(* ---------------------------------------------------------
   Z轴External纯轨迹发生器。
   进入：External Adapter已Active且已接受P/V/A/Direction有效。
   周期动作：只从最后accepted包进行Rate Limit和梯形积分。
   换向：零速、旧方向保持、方向归零、新方向预置均由accepted Feed推进。
   硬禁止：同一扫描保持accepted位置并发布V=0、A=0、方向不变。
   Fault：首次故障锁存；调用者必须停止Feed并请求Adapter安全Disable。
   --------------------------------------------------------- *)
stOutput.rPosition_mm := 0.0;
stOutput.rVelocity_mm_s := 0.0;
stOutput.rAcceleration_mm_s2 := 0.0;
stOutput.nDirection := 0;
stOutput.eState := eState;
stOutput.bDirectionTransition := FALSE;
stOutput.bZeroConfirmed := FALSE;
stOutput.bPositiveMotionInhibited := FALSE;
stOutput.bActive := FALSE;
stOutput.bFault := bFaultLatched;
stOutput.nFaultId := udiLatchedFaultId;

(* Fault只能在未使能时显式复位；复位扫描保持IDLE和非活动。 *)
IF bFaultLatched THEN
    eState := Z_TRAJ_FAULT;
    stOutput.eState := Z_TRAJ_FAULT;
    stOutput.bActive := FALSE;
    stOutput.bFault := TRUE;
    stOutput.nFaultId := udiLatchedFaultId;
    IF stInput.bReset AND NOT stInput.bEnable THEN
        bFaultLatched := FALSE;
        udiLatchedFaultId := 0;
        bInitialized := FALSE;
        bLastPublishedPositiveMotionInhibited := FALSE;
        udiLastAcceptedFeedCycleCounter := 0;
        nLastNonZeroDirection := 0;
        nPendingDirection := 0;
        nAcceptedStateCycles := 0;
        eState := Z_TRAJ_IDLE;
        stOutput.bFault := FALSE;
        stOutput.nFaultId := 0;
        stOutput.bActive := FALSE;
        stOutput.eState := Z_TRAJ_IDLE;
    END_IF;
    RETURN;
END_IF;

(* Disable清除运行态但不伪造Active或轨迹Feed。 *)
IF NOT stInput.bEnable THEN
    bInitialized := FALSE;
    bLastPublishedPositiveMotionInhibited := FALSE;
    udiLastAcceptedFeedCycleCounter := 0;
    nLastNonZeroDirection := 0;
    nPendingDirection := 0;
    nAcceptedStateCycles := 0;
    eState := Z_TRAJ_IDLE;
    stOutput.eState := Z_TRAJ_IDLE;
    RETURN;
END_IF;

nTargetDirection := 0;
IF stInput.rTargetVelocity_mm_s > 0.0 THEN
    nTargetDirection := 1;
ELSIF stInput.rTargetVelocity_mm_s < 0.0 THEN
    nTargetDirection := -1;
END_IF;

bConfigurationValid := (stInput.rCycleTime_s > 0.0)
    AND FC_IsFiniteLReal(rValue := stInput.rCycleTime_s)
    AND FC_IsFiniteLReal(rValue := stInput.rMinimumPosition_mm)
    AND FC_IsFiniteLReal(rValue := stInput.rMaximumPosition_mm)
    AND (stInput.rMaximumPosition_mm > stInput.rMinimumPosition_mm)
    AND FC_IsFiniteLReal(rValue := stInput.rMaximumVelocity_mm_s)
    AND (stInput.rMaximumVelocity_mm_s > 0.0)
    AND FC_IsFiniteLReal(rValue := stInput.rMaximumAcceleration_mm_s2)
    AND (stInput.rMaximumAcceleration_mm_s2 > 0.0)
    AND FC_IsFiniteLReal(rValue := stInput.rStandstillVelocity_mm_s)
    AND (stInput.rStandstillVelocity_mm_s >= 0.0)
    AND (stInput.rStandstillVelocity_mm_s < stInput.rMaximumVelocity_mm_s)
    AND FC_IsFiniteLReal(rValue := stInput.rMaximumPositionDeviation_mm)
    AND (stInput.rMaximumPositionDeviation_mm >= 0.0)
    AND FC_IsFiniteLReal(rValue := stInput.rTargetVelocity_mm_s)
    AND (ABS(stInput.rTargetVelocity_mm_s) <= stInput.rMaximumVelocity_mm_s)
    AND (stInput.nDirectionHoldCycles >= 1);

IF NOT bConfigurationValid THEN
    bFaultLatched := TRUE;
    udiLatchedFaultId := 16#0000B001;
    eState := Z_TRAJ_FAULT;
    stOutput.bFault := TRUE;
    stOutput.nFaultId := udiLatchedFaultId;
    stOutput.eState := Z_TRAJ_FAULT;
    stOutput.bActive := FALSE;
    RETURN;
END_IF;

(* Adapter未Active时只等待重新同步，不消费或外推任何包。 *)
IF stInput.eExternalState <> Z_EXT_ACTIVE THEN
    bInitialized := FALSE;
    bLastPublishedPositiveMotionInhibited := FALSE;
    nAcceptedStateCycles := 0;
    eState := Z_TRAJ_SYNC;
    stOutput.eState := Z_TRAJ_SYNC;
    RETURN;
END_IF;

bAcceptedMotionValid := stInput.bAcceptedSetpointValid
    AND FC_IsFiniteLReal(rValue := stInput.rAcceptedPosition_mm)
    AND FC_IsFiniteLReal(rValue := stInput.rAcceptedVelocity_mm_s)
    AND FC_IsFiniteLReal(rValue := stInput.rAcceptedAcceleration_mm_s2)
    AND (ABS(stInput.rAcceptedVelocity_mm_s) <= stInput.rMaximumVelocity_mm_s)
    AND (ABS(stInput.rAcceptedAcceleration_mm_s2) <= stInput.rMaximumAcceleration_mm_s2);

IF NOT bAcceptedMotionValid THEN
    bFaultLatched := TRUE;
    udiLatchedFaultId := 16#0000B002;
    eState := Z_TRAJ_FAULT;
    stOutput.bFault := TRUE;
    stOutput.nFaultId := udiLatchedFaultId;
    stOutput.eState := Z_TRAJ_FAULT;
    stOutput.bActive := FALSE;
    RETURN;
END_IF;

IF (stInput.nAcceptedDirection < -1) OR (stInput.nAcceptedDirection > 1) THEN
    bFaultLatched := TRUE;
    udiLatchedFaultId := 16#0000B003;
    eState := Z_TRAJ_FAULT;
    stOutput.bFault := TRUE;
    stOutput.nFaultId := udiLatchedFaultId;
    stOutput.eState := Z_TRAJ_FAULT;
    stOutput.bActive := FALSE;
    RETURN;
END_IF;

IF (stInput.rAcceptedPosition_mm < stInput.rMinimumPosition_mm)
    OR (stInput.rAcceptedPosition_mm > stInput.rMaximumPosition_mm) THEN
    bFaultLatched := TRUE;
    udiLatchedFaultId := 16#0000B004;
    eState := Z_TRAJ_FAULT;
    stOutput.bFault := TRUE;
    stOutput.nFaultId := udiLatchedFaultId;
    stOutput.eState := Z_TRAJ_FAULT;
    stOutput.bActive := FALSE;
    RETURN;
END_IF;

IF (stInput.nAcceptedDirection = 0)
    AND ((ABS(stInput.rAcceptedVelocity_mm_s) > stInput.rStandstillVelocity_mm_s)
        OR (stInput.rAcceptedAcceleration_mm_s2 <> 0.0)) THEN
    bFaultLatched := TRUE;
    udiLatchedFaultId := 16#0000B007;
    eState := Z_TRAJ_FAULT;
    stOutput.bFault := TRUE;
    stOutput.nFaultId := udiLatchedFaultId;
    stOutput.eState := Z_TRAJ_FAULT;
    stOutput.bActive := FALSE;
    RETURN;
END_IF;

IF ((stInput.rAcceptedVelocity_mm_s > stInput.rStandstillVelocity_mm_s)
        AND (stInput.nAcceptedDirection <> 1))
    OR ((stInput.rAcceptedVelocity_mm_s < -stInput.rStandstillVelocity_mm_s)
        AND (stInput.nAcceptedDirection <> -1)) THEN
    bFaultLatched := TRUE;
    udiLatchedFaultId := 16#0000B006;
    eState := Z_TRAJ_FAULT;
    stOutput.bFault := TRUE;
    stOutput.nFaultId := udiLatchedFaultId;
    stOutput.eState := Z_TRAJ_FAULT;
    stOutput.bActive := FALSE;
    RETURN;
END_IF;

bNewAcceptedFeed := (stInput.bFeedAccepted = TRUE)
    AND (stInput.udiAcceptedFeedCycleCounter <> udiLastAcceptedFeedCycleCounter);
bAcceptedPublishedZero := FALSE;
stOutput.bPositiveMotionInhibited := stInput.bInhibitPositiveMotion;

IF NOT bInitialized THEN
    (* 首个Active扫描只发布同步包；必须等该包accepted后才进入TRACKING。 *)
    udiLastAcceptedFeedCycleCounter := stInput.udiAcceptedFeedCycleCounter;
    IF stInput.nAcceptedDirection <> 0 THEN
        nLastNonZeroDirection := stInput.nAcceptedDirection;
    END_IF;
    bInitialized := TRUE;
    eState := Z_TRAJ_SYNC;
    stOutput.eState := Z_TRAJ_SYNC;
    stOutput.rPosition_mm := stInput.rAcceptedPosition_mm;
    stOutput.rVelocity_mm_s := stInput.rAcceptedVelocity_mm_s;
    stOutput.rAcceleration_mm_s2 := stInput.rAcceptedAcceleration_mm_s2;
    stOutput.nDirection := stInput.nAcceptedDirection;
    IF stInput.bInhibitPositiveMotion
        AND (stInput.rAcceptedVelocity_mm_s > 0.0) THEN
        stOutput.rPosition_mm := stInput.rAcceptedPosition_mm;
        stOutput.rVelocity_mm_s := 0.0;
        stOutput.rAcceleration_mm_s2 := 0.0;
        stOutput.nDirection := stInput.nAcceptedDirection;
        stOutput.bPositiveMotionInhibited := TRUE;
    END_IF;
    rLastPublishedPosition_mm := stOutput.rPosition_mm;
    rLastPublishedVelocity_mm_s := stOutput.rVelocity_mm_s;
    rLastPublishedAcceleration_mm_s2 := stOutput.rAcceleration_mm_s2;
    nLastPublishedDirection := stOutput.nDirection;
    bLastPublishedPositiveMotionInhibited := stOutput.bPositiveMotionInhibited;
    stOutput.bActive := TRUE;
    RETURN;
ELSE
    IF bNewAcceptedFeed THEN
        IF (stInput.nAcceptedDirection <> nLastPublishedDirection)
            AND (ABS(stInput.rAcceptedVelocity_mm_s) > stInput.rStandstillVelocity_mm_s) THEN
            bFaultLatched := TRUE;
            udiLatchedFaultId := 16#0000B006;
            eState := Z_TRAJ_FAULT;
            stOutput.bFault := TRUE;
            stOutput.nFaultId := udiLatchedFaultId;
            stOutput.eState := Z_TRAJ_FAULT;
            stOutput.bActive := FALSE;
            RETURN;
        END_IF;
        IF (eState <> Z_TRAJ_PRELOAD_NEW_DIRECTION)
            AND (stInput.nAcceptedDirection <> 0)
            AND (nLastNonZeroDirection <> 0)
            AND (stInput.nAcceptedDirection <> nLastNonZeroDirection) THEN
            bFaultLatched := TRUE;
            udiLatchedFaultId := 16#0000B006;
            eState := Z_TRAJ_FAULT;
            stOutput.bFault := TRUE;
            stOutput.nFaultId := udiLatchedFaultId;
            stOutput.eState := Z_TRAJ_FAULT;
            stOutput.bActive := FALSE;
            RETURN;
        END_IF;

        bAcceptedContinuityValid := ABS(stInput.rAcceptedPosition_mm
                - rLastPublishedPosition_mm) <= stInput.rMaximumPositionDeviation_mm
            AND (stInput.rAcceptedVelocity_mm_s = rLastPublishedVelocity_mm_s)
            AND (stInput.rAcceptedAcceleration_mm_s2 = rLastPublishedAcceleration_mm_s2)
            AND (stInput.nAcceptedDirection = nLastPublishedDirection);
        IF NOT bAcceptedContinuityValid THEN
            bFaultLatched := TRUE;
            udiLatchedFaultId := 16#0000B005;
            eState := Z_TRAJ_FAULT;
            stOutput.bFault := TRUE;
            stOutput.nFaultId := udiLatchedFaultId;
            stOutput.eState := Z_TRAJ_FAULT;
            stOutput.bActive := FALSE;
            RETURN;
        END_IF;

        bAcceptedPublishedZero := (rLastPublishedVelocity_mm_s = 0.0)
            AND (rLastPublishedAcceleration_mm_s2 = 0.0)
            AND (ABS(stInput.rAcceptedVelocity_mm_s) <= stInput.rStandstillVelocity_mm_s)
            AND (stInput.rAcceptedAcceleration_mm_s2 = 0.0);
        udiLastAcceptedFeedCycleCounter := stInput.udiAcceptedFeedCycleCounter;
        IF stInput.nAcceptedDirection <> 0 THEN
            nLastNonZeroDirection := stInput.nAcceptedDirection;
        END_IF;
    END_IF;
END_IF;

stOutput.bZeroConfirmed := bNewAcceptedFeed AND bAcceptedPublishedZero;

(* 转换期间目标方向必须保持为进入转换时锁存的非零方向。 *)
IF (eState = Z_TRAJ_RAMP_TO_ZERO)
    OR (eState = Z_TRAJ_HOLD_OLD_DIRECTION)
    OR (eState = Z_TRAJ_DIRECTION_ZERO)
    OR (eState = Z_TRAJ_PRELOAD_NEW_DIRECTION) THEN
    IF (nTargetDirection = 0) OR (nTargetDirection <> nPendingDirection) THEN
        bFaultLatched := TRUE;
        udiLatchedFaultId := 16#0000B00A;
        eState := Z_TRAJ_FAULT;
        stOutput.bFault := TRUE;
        stOutput.nFaultId := udiLatchedFaultId;
        stOutput.eState := Z_TRAJ_FAULT;
        stOutput.bActive := FALSE;
        RETURN;
    END_IF;
END_IF;

stOutput.eState := eState;
stOutput.bDirectionTransition := (eState = Z_TRAJ_RAMP_TO_ZERO)
    OR (eState = Z_TRAJ_HOLD_OLD_DIRECTION)
    OR (eState = Z_TRAJ_DIRECTION_ZERO)
    OR (eState = Z_TRAJ_PRELOAD_NEW_DIRECTION);

(* Hard Inhibit是唯一允许替换未接受普通包的安全优先级。 *)
IF NOT bNewAcceptedFeed AND stInput.bInhibitPositiveMotion
    AND ((stInput.rAcceptedVelocity_mm_s > 0.0)
        OR (rLastPublishedVelocity_mm_s > 0.0)) THEN
    stOutput.rPosition_mm := stInput.rAcceptedPosition_mm;
    stOutput.rVelocity_mm_s := 0.0;
    stOutput.rAcceleration_mm_s2 := 0.0;
    stOutput.nDirection := stInput.nAcceptedDirection;
    stOutput.bPositiveMotionInhibited := TRUE;
    rLastPublishedPosition_mm := stOutput.rPosition_mm;
    rLastPublishedVelocity_mm_s := stOutput.rVelocity_mm_s;
    rLastPublishedAcceleration_mm_s2 := stOutput.rAcceleration_mm_s2;
    nLastPublishedDirection := stOutput.nDirection;
    bLastPublishedPositiveMotionInhibited := stOutput.bPositiveMotionInhibited;
    stOutput.bActive := TRUE;
    RETURN;
END_IF;

(* 无新accepted counter时严格重复待接受包，忽略TRACKING实时目标变化。 *)
IF NOT bNewAcceptedFeed THEN
    stOutput.rPosition_mm := rLastPublishedPosition_mm;
    stOutput.rVelocity_mm_s := rLastPublishedVelocity_mm_s;
    stOutput.rAcceleration_mm_s2 := rLastPublishedAcceleration_mm_s2;
    stOutput.nDirection := nLastPublishedDirection;
    stOutput.bPositiveMotionInhibited := bLastPublishedPositiveMotionInhibited;
    stOutput.bActive := TRUE;
    RETURN;
END_IF;

CASE eState OF
    Z_TRAJ_IDLE:
        eState := Z_TRAJ_SYNC;

    Z_TRAJ_SYNC:
        (* 同步扫描原样发布accepted包，下一扫描才开始积分。 *)
        stOutput.rPosition_mm := stInput.rAcceptedPosition_mm;
        stOutput.rVelocity_mm_s := stInput.rAcceptedVelocity_mm_s;
        stOutput.rAcceleration_mm_s2 := stInput.rAcceptedAcceleration_mm_s2;
        stOutput.nDirection := stInput.nAcceptedDirection;
        IF bInitialized THEN
            eState := Z_TRAJ_TRACKING;
        END_IF;

    Z_TRAJ_TRACKING:
        IF (nTargetDirection <> 0)
            AND (nLastNonZeroDirection <> 0)
            AND (nTargetDirection <> nLastNonZeroDirection) THEN
            (* 非零反向目标先按accepted速度主动降到零。 *)
            nPendingDirection := nTargetDirection;
            nAcceptedStateCycles := 0;
            eState := Z_TRAJ_RAMP_TO_ZERO;
            rNextVelocity_mm_s := FC_LimitRate(
                rCurrent := stInput.rAcceptedVelocity_mm_s,
                rTarget := 0.0,
                rRateUpPer_s := stInput.rMaximumAcceleration_mm_s2,
                rRateDownPer_s := stInput.rMaximumAcceleration_mm_s2,
                rCycleTime_s := stInput.rCycleTime_s);
            rNextAcceleration_mm_s2 :=
                (rNextVelocity_mm_s - stInput.rAcceptedVelocity_mm_s)
                / stInput.rCycleTime_s;
            rNextPosition_mm := stInput.rAcceptedPosition_mm
                + 0.5 * (stInput.rAcceptedVelocity_mm_s + rNextVelocity_mm_s)
                * stInput.rCycleTime_s;
            stOutput.rPosition_mm := rNextPosition_mm;
            stOutput.rVelocity_mm_s := rNextVelocity_mm_s;
            stOutput.rAcceleration_mm_s2 := rNextAcceleration_mm_s2;
            stOutput.nDirection := nLastNonZeroDirection;
        ELSIF (stInput.nAcceptedDirection = 0) AND (nTargetDirection <> 0) THEN
            (* 静止初始状态先预置新方向一个被接受的完整周期。 *)
            nPendingDirection := nTargetDirection;
            nAcceptedStateCycles := 0;
            eState := Z_TRAJ_PRELOAD_NEW_DIRECTION;
            stOutput.rPosition_mm := stInput.rAcceptedPosition_mm;
            stOutput.rVelocity_mm_s := 0.0;
            stOutput.rAcceleration_mm_s2 := 0.0;
            stOutput.nDirection := nPendingDirection;
        ELSE
            rNextVelocity_mm_s := FC_LimitRate(
                rCurrent := stInput.rAcceptedVelocity_mm_s,
                rTarget := stInput.rTargetVelocity_mm_s,
                rRateUpPer_s := stInput.rMaximumAcceleration_mm_s2,
                rRateDownPer_s := stInput.rMaximumAcceleration_mm_s2,
                rCycleTime_s := stInput.rCycleTime_s);
            IF stInput.bInhibitPositiveMotion AND (rNextVelocity_mm_s > 0.0) THEN
                rNextVelocity_mm_s := 0.0;
            END_IF;
            rNextAcceleration_mm_s2 :=
                (rNextVelocity_mm_s - stInput.rAcceptedVelocity_mm_s)
                / stInput.rCycleTime_s;
            rNextPosition_mm := stInput.rAcceptedPosition_mm
                + 0.5 * (stInput.rAcceptedVelocity_mm_s + rNextVelocity_mm_s)
                * stInput.rCycleTime_s;
            stOutput.rPosition_mm := rNextPosition_mm;
            stOutput.rVelocity_mm_s := rNextVelocity_mm_s;
            stOutput.rAcceleration_mm_s2 := rNextAcceleration_mm_s2;
            stOutput.nDirection := stInput.nAcceptedDirection;
        END_IF;

        (* Hard Force/Stroke/Collision覆盖普通正向制动尾巴。 *)
        IF stInput.bInhibitPositiveMotion THEN
            IF stInput.rAcceptedVelocity_mm_s > 0.0 THEN
                stOutput.rPosition_mm := stInput.rAcceptedPosition_mm;
                stOutput.rVelocity_mm_s := 0.0;
                stOutput.rAcceleration_mm_s2 := 0.0;
                stOutput.nDirection := stInput.nAcceptedDirection;
                stOutput.bPositiveMotionInhibited := TRUE;
            ELSIF stOutput.rVelocity_mm_s > 0.0 THEN
                stOutput.rPosition_mm := stInput.rAcceptedPosition_mm;
                stOutput.rVelocity_mm_s := 0.0;
                stOutput.rAcceleration_mm_s2 := 0.0;
                stOutput.nDirection := stInput.nAcceptedDirection;
                stOutput.bPositiveMotionInhibited := TRUE;
            ELSE
                stOutput.bPositiveMotionInhibited := TRUE;
            END_IF;
        END_IF;

    Z_TRAJ_RAMP_TO_ZERO:
        rNextVelocity_mm_s := FC_LimitRate(
            rCurrent := stInput.rAcceptedVelocity_mm_s,
            rTarget := 0.0,
            rRateUpPer_s := stInput.rMaximumAcceleration_mm_s2,
            rRateDownPer_s := stInput.rMaximumAcceleration_mm_s2,
            rCycleTime_s := stInput.rCycleTime_s);
        IF ABS(rNextVelocity_mm_s) <= stInput.rStandstillVelocity_mm_s THEN
            rNextVelocity_mm_s := 0.0;
        END_IF;
        rNextAcceleration_mm_s2 :=
            (rNextVelocity_mm_s - stInput.rAcceptedVelocity_mm_s)
            / stInput.rCycleTime_s;
        rNextPosition_mm := stInput.rAcceptedPosition_mm
            + 0.5 * (stInput.rAcceptedVelocity_mm_s + rNextVelocity_mm_s)
            * stInput.rCycleTime_s;
        stOutput.rPosition_mm := rNextPosition_mm;
        stOutput.rVelocity_mm_s := rNextVelocity_mm_s;
        stOutput.rAcceleration_mm_s2 := rNextAcceleration_mm_s2;
        stOutput.nDirection := nLastNonZeroDirection;
        IF stInput.bInhibitPositiveMotion AND (stInput.rAcceptedVelocity_mm_s > 0.0) THEN
            stOutput.rPosition_mm := stInput.rAcceptedPosition_mm;
            stOutput.rVelocity_mm_s := 0.0;
            stOutput.rAcceleration_mm_s2 := 0.0;
            stOutput.nDirection := stInput.nAcceptedDirection;
            stOutput.bPositiveMotionInhibited := TRUE;
        END_IF;
        IF stOutput.bZeroConfirmed THEN
            nAcceptedStateCycles := 0;
            eState := Z_TRAJ_HOLD_OLD_DIRECTION;
        END_IF;

    Z_TRAJ_HOLD_OLD_DIRECTION:
        stOutput.rPosition_mm := stInput.rAcceptedPosition_mm;
        stOutput.rVelocity_mm_s := 0.0;
        stOutput.rAcceleration_mm_s2 := 0.0;
        stOutput.nDirection := nLastNonZeroDirection;
        IF bNewAcceptedFeed THEN
            IF nAcceptedStateCycles < UINT#65535 THEN
                nAcceptedStateCycles := nAcceptedStateCycles + 1;
            END_IF;
            IF nAcceptedStateCycles >= stInput.nDirectionHoldCycles THEN
                nAcceptedStateCycles := 0;
                eState := Z_TRAJ_DIRECTION_ZERO;
            END_IF;
        END_IF;

    Z_TRAJ_DIRECTION_ZERO:
        stOutput.rPosition_mm := stInput.rAcceptedPosition_mm;
        stOutput.rVelocity_mm_s := 0.0;
        stOutput.rAcceleration_mm_s2 := 0.0;
        stOutput.nDirection := 0;
        IF bNewAcceptedFeed AND (stInput.nAcceptedDirection = 0) THEN
            nAcceptedStateCycles := 0;
            eState := Z_TRAJ_PRELOAD_NEW_DIRECTION;
        END_IF;

    Z_TRAJ_PRELOAD_NEW_DIRECTION:
        stOutput.rPosition_mm := stInput.rAcceptedPosition_mm;
        stOutput.rVelocity_mm_s := 0.0;
        stOutput.rAcceleration_mm_s2 := 0.0;
        stOutput.nDirection := nPendingDirection;
        IF bNewAcceptedFeed
            AND (stInput.nAcceptedDirection = nPendingDirection) THEN
            nLastNonZeroDirection := nPendingDirection;
            nAcceptedStateCycles := 0;
            eState := Z_TRAJ_TRACKING;
        END_IF;

    Z_TRAJ_FAULT:
        stOutput.rPosition_mm := stInput.rAcceptedPosition_mm;
        stOutput.rVelocity_mm_s := 0.0;
        stOutput.rAcceleration_mm_s2 := 0.0;
        stOutput.nDirection := stInput.nAcceptedDirection;
        stOutput.bFault := TRUE;
        stOutput.nFaultId := udiLatchedFaultId;
        stOutput.bActive := FALSE;
        IF stInput.bReset AND NOT stInput.bEnable THEN
            bFaultLatched := FALSE;
            udiLatchedFaultId := 0;
            bInitialized := FALSE;
            bLastPublishedPositiveMotionInhibited := FALSE;
            eState := Z_TRAJ_IDLE;
            stOutput.bFault := FALSE;
            stOutput.nFaultId := 0;
            stOutput.bActive := FALSE;
            stOutput.eState := Z_TRAJ_IDLE;
        END_IF;

ELSE
    bFaultLatched := TRUE;
    udiLatchedFaultId := 16#0000B009;
    eState := Z_TRAJ_FAULT;
    stOutput.bFault := TRUE;
    stOutput.nFaultId := udiLatchedFaultId;
    stOutput.eState := Z_TRAJ_FAULT;
    stOutput.bActive := FALSE;
    RETURN;
END_CASE;

(* 所有Active状态统一执行Hard Inhibit，消除SYNC和转换态的正向尾包。 *)
IF stInput.bInhibitPositiveMotion
    AND (stInput.rAcceptedVelocity_mm_s > 0.0) THEN
    stOutput.rPosition_mm := stInput.rAcceptedPosition_mm;
    stOutput.rVelocity_mm_s := 0.0;
    stOutput.rAcceleration_mm_s2 := 0.0;
    stOutput.nDirection := stInput.nAcceptedDirection;
    stOutput.bPositiveMotionInhibited := TRUE;
ELSIF stInput.bInhibitPositiveMotion
    AND (stOutput.rVelocity_mm_s > 0.0) THEN
    stOutput.rPosition_mm := stInput.rAcceptedPosition_mm;
    stOutput.rVelocity_mm_s := 0.0;
    stOutput.rAcceleration_mm_s2 := 0.0;
    stOutput.nDirection := stInput.nAcceptedDirection;
    stOutput.bPositiveMotionInhibited := TRUE;
END_IF;

IF (stOutput.rPosition_mm < stInput.rMinimumPosition_mm)
    OR (stOutput.rPosition_mm > stInput.rMaximumPosition_mm)
    OR NOT FC_IsFiniteLReal(rValue := stOutput.rPosition_mm) THEN
    bFaultLatched := TRUE;
    udiLatchedFaultId := 16#0000B008;
    eState := Z_TRAJ_FAULT;
    stOutput.bFault := TRUE;
    stOutput.nFaultId := udiLatchedFaultId;
    stOutput.eState := Z_TRAJ_FAULT;
    stOutput.bActive := FALSE;
    RETURN;
END_IF;

stOutput.eState := eState;
stOutput.bDirectionTransition := (eState = Z_TRAJ_RAMP_TO_ZERO)
    OR (eState = Z_TRAJ_HOLD_OLD_DIRECTION)
    OR (eState = Z_TRAJ_DIRECTION_ZERO)
    OR (eState = Z_TRAJ_PRELOAD_NEW_DIRECTION);
stOutput.bActive := (stInput.eExternalState = Z_EXT_ACTIVE)
    AND ((eState = Z_TRAJ_SYNC)
        OR (eState = Z_TRAJ_TRACKING)
        OR (eState = Z_TRAJ_RAMP_TO_ZERO)
        OR (eState = Z_TRAJ_HOLD_OLD_DIRECTION)
        OR (eState = Z_TRAJ_DIRECTION_ZERO)
        OR (eState = Z_TRAJ_PRELOAD_NEW_DIRECTION));

(* 仅保存本扫描实际发布包；下一扫描先验证accepted，再生成后续包。 *)
rLastPublishedPosition_mm := stOutput.rPosition_mm;
rLastPublishedVelocity_mm_s := stOutput.rVelocity_mm_s;
rLastPublishedAcceleration_mm_s2 := stOutput.rAcceleration_mm_s2;
nLastPublishedDirection := stOutput.nDirection;
bLastPublishedPositiveMotionInhibited := stOutput.bPositiveMotionInhibited;

END_FUNCTION_BLOCK

// ---- POUs/FunctionBlocks/Axis/FB_ZAxisNcAdapter.TcPOU
FUNCTION_BLOCK FB_ZAxisNcAdapter
VAR_IN_OUT
    (* 唯一Z轴NC引用；仅允许本Adapter访问。 *)
    Axis : AXIS_REF;
END_VAR
VAR_INPUT
    (* 真实驱动、编码器和NC轴已经人工关联并验证。 *)
    bDriveLinked : BOOL;
    (* 上层命令事务编号；只有变化才产生MC Execute上升沿。 *)
    udiCommandId : UDINT;
    (* 经Owner仲裁的唯一Z轴标准命令。 *)
    stCommand : ST_ZAxisCommand;
END_VAR
VAR_OUTPUT
    (* Z轴标准运动状态快照。 *)
    stStatus : ST_ZAxisStatus;
    (* Adapter已处理的最后命令事务编号。 *)
    udiAcceptedCommandId : UDINT;
END_VAR
VAR
    (* Z轴软件使能实例。 *)
    fbPower : MC_Power;
    (* Z轴错误复位实例。 *)
    fbReset : MC_Reset;
    (* Z轴标准回零实例。 *)
    fbHome : MC_Home;
    (* Z轴绝对定位实例。 *)
    fbMoveAbsolute : MC_MoveAbsolute;
    (* Z轴速度运动双实例A，用于以新命令替换活动速度命令。 *)
    fbMoveVelocityA : MC_MoveVelocity;
    (* Z轴速度运动双实例B，用于以新命令替换活动速度命令。 *)
    fbMoveVelocityB : MC_MoveVelocity;
    (* Z轴受控停止实例。 *)
    fbHalt : MC_Halt;
    (* 当前扫描检测到新的命令编号。 *)
    bNewCommand : BOOL;
    (* 当前扫描的复位Execute脉冲。 *)
    bResetPulse : BOOL;
    (* 当前扫描的回零Execute脉冲。 *)
    bHomePulse : BOOL;
    (* 当前扫描的绝对定位Execute脉冲。 *)
    bMoveAbsolutePulse : BOOL;
    (* 当前扫描速度实例A的Execute脉冲。 *)
    bMoveVelocityPulseA : BOOL;
    (* 当前扫描速度实例B的Execute脉冲。 *)
    bMoveVelocityPulseB : BOOL;
    (* 当前扫描的受控停止Execute脉冲。 *)
    bHaltPulse : BOOL;
    (* 下次速度命令选择A实例，否则选择B实例。 *)
    bSelectVelocityA : BOOL;
    (* 速度命令方向。 *)
    eVelocityDirection : MC_Direction;
END_VAR

(* ---------------------------------------------------------
   Z轴标准NC Adapter状态。
   进入：Task_CffFast每扫描调用，且由PRG_FastAxisControl唯一持有。
   动作：更新AXIS_REF状态；命令编号变化时产生一次MC上升沿。
   成功：发布真实NC状态；Ready还必须满足真实驱动已人工关联。
   超时：由上层流程负责；MC Busy/Error保持可诊断。
   Fault：Stop优先；未绑定驱动时Power和全部运动Execute硬门控。
   --------------------------------------------------------- *)
Axis.ReadStatus();

bNewCommand := udiCommandId <> udiAcceptedCommandId;
bResetPulse := FALSE;
bHomePulse := FALSE;
bMoveAbsolutePulse := FALSE;
bMoveVelocityPulseA := FALSE;
bMoveVelocityPulseB := FALSE;
bHaltPulse := FALSE;

IF stCommand.rVelocity_mm_s >= 0.0 THEN
    eVelocityDirection := MC_Positive_Direction;
ELSE
    eVelocityDirection := MC_Negative_Direction;
END_IF

IF bNewCommand THEN
    udiAcceptedCommandId := udiCommandId;
    bResetPulse := bDriveLinked AND stCommand.bReset;

    IF bDriveLinked AND stCommand.bStop THEN
        bHaltPulse := TRUE;
    ELSIF bDriveLinked AND stCommand.bEnable AND NOT stCommand.bUseExternalSetpoint THEN
        IF stCommand.bHome THEN
            bHomePulse := TRUE;
        ELSIF stCommand.bMoveAbsolute THEN
            bMoveAbsolutePulse := TRUE;
        ELSIF stCommand.bMoveVelocity THEN
            IF ABS(stCommand.rVelocity_mm_s) > 0.0 THEN
                bSelectVelocityA := NOT bSelectVelocityA;
                bMoveVelocityPulseA := bSelectVelocityA;
                bMoveVelocityPulseB := NOT bSelectVelocityA;
            ELSE
                bHaltPulse := TRUE;
            END_IF
        END_IF
    END_IF
END_IF

(* 未完成真实驱动关联时Enable恒为FALSE，不能因离线NC对象而产生Ready。 *)
fbPower(
    Axis := Axis,
    Enable := bDriveLinked AND stCommand.bEnable,
    Enable_Positive := bDriveLinked AND stCommand.bEnable,
    Enable_Negative := bDriveLinked AND stCommand.bEnable,
    Override := 100.0,
    BufferMode := MC_Aborting);
fbReset(Axis := Axis, Execute := bResetPulse);
fbHome(
    Axis := Axis,
    Execute := bHomePulse,
    Position := stCommand.rHomePosition_mm,
    HomingMode := MC_DefaultHoming);
fbMoveAbsolute(
    Axis := Axis,
    Execute := bMoveAbsolutePulse,
    Position := stCommand.rPosition_mm,
    Velocity := ABS(stCommand.rVelocity_mm_s),
    Acceleration := ABS(stCommand.rAcceleration_mm_s2),
    Deceleration := ABS(stCommand.rDeceleration_mm_s2),
    Jerk := 0.0,
    BufferMode := MC_Aborting);
fbMoveVelocityA(
    Axis := Axis,
    Execute := bMoveVelocityPulseA,
    Velocity := ABS(stCommand.rVelocity_mm_s),
    Acceleration := ABS(stCommand.rAcceleration_mm_s2),
    Deceleration := ABS(stCommand.rDeceleration_mm_s2),
    Jerk := 0.0,
    Direction := eVelocityDirection,
    BufferMode := MC_Aborting);
fbMoveVelocityB(
    Axis := Axis,
    Execute := bMoveVelocityPulseB,
    Velocity := ABS(stCommand.rVelocity_mm_s),
    Acceleration := ABS(stCommand.rAcceleration_mm_s2),
    Deceleration := ABS(stCommand.rDeceleration_mm_s2),
    Jerk := 0.0,
    Direction := eVelocityDirection,
    BufferMode := MC_Aborting);
fbHalt(
    Axis := Axis,
    Execute := bHaltPulse,
    Deceleration := ABS(stCommand.rDeceleration_mm_s2),
    Jerk := 0.0,
    BufferMode := MC_Aborting);

stStatus.bError := bDriveLinked AND (Axis.Status.Error OR fbPower.Error OR fbReset.Error
    OR fbHome.Error OR fbMoveAbsolute.Error OR fbMoveVelocityA.Error
    OR fbMoveVelocityB.Error OR fbHalt.Error);
stStatus.nErrorId := 0;
IF bDriveLinked AND Axis.Status.Error THEN
    stStatus.nErrorId := DWORD_TO_UDINT(Axis.NcToPlc.ErrorCode);
ELSIF fbPower.Error THEN
    stStatus.nErrorId := fbPower.ErrorID;
ELSIF fbReset.Error THEN
    stStatus.nErrorId := fbReset.ErrorID;
ELSIF fbHome.Error THEN
    stStatus.nErrorId := fbHome.ErrorID;
ELSIF fbMoveAbsolute.Error THEN
    stStatus.nErrorId := fbMoveAbsolute.ErrorID;
ELSIF fbMoveVelocityA.Error THEN
    stStatus.nErrorId := fbMoveVelocityA.ErrorID;
ELSIF fbMoveVelocityB.Error THEN
    stStatus.nErrorId := fbMoveVelocityB.ErrorID;
ELSIF fbHalt.Error THEN
    stStatus.nErrorId := fbHalt.ErrorID;
END_IF

stStatus.bReady := bDriveLinked AND fbPower.Status AND Axis.Status.Operational
    AND NOT stStatus.bError;
stStatus.bEnabled := bDriveLinked AND fbPower.Status;
stStatus.bHomed := bDriveLinked AND Axis.Status.Homed;
stStatus.bMoving := bDriveLinked AND (Axis.Status.DiscreteMotion
    OR Axis.Status.ContinuousMotion OR Axis.Status.Homing);
stStatus.bStandstill := bDriveLinked AND Axis.Status.StandStill;
stStatus.bBusy := bDriveLinked AND (fbReset.Busy OR fbHome.Busy OR fbMoveAbsolute.Busy
    OR fbMoveVelocityA.Busy OR fbMoveVelocityB.Busy OR fbHalt.Busy);
stStatus.bDone := bDriveLinked AND (fbReset.Done OR fbHome.Done OR fbMoveAbsolute.Done
    OR fbMoveVelocityA.InVelocity OR fbMoveVelocityB.InVelocity OR fbHalt.Done);
stStatus.bExternalSetpointActive := FALSE;
stStatus.eActiveOwner := stCommand.eOwnerRequest;
stStatus.udiAcceptedCommandId := udiAcceptedCommandId;

IF bDriveLinked THEN
    stStatus.rActualPosition_mm := Axis.NcToPlc.ActPos;
    stStatus.rActualVelocity_mm_s := Axis.NcToPlc.ActVelo;
ELSE
    stStatus.rActualPosition_mm := 0.0;
    stStatus.rActualVelocity_mm_s := 0.0;
END_IF;

END_FUNCTION_BLOCK

// ---- POUs/FunctionBlocks/Axis/FB_ZAxisExtSetpointAdapter.TcPOU
FUNCTION_BLOCK FB_ZAxisExtSetpointAdapter
VAR_IN_OUT
    (* 唯一Z轴NC引用；只通过Tc2_MC2 External Setpoint接口访问。 *)
    Axis : AXIS_REF;
END_VAR
VAR_INPUT
    (* 真实驱动、编码器和NC轴已经人工关联并验证。 *)
    bDriveLinked : BOOL;
    (* Z轴Owner已经由仲裁器授予Force Process。 *)
    bOwnerGranted : BOOL;
    (* 机器Z轴硬限值集合已经受控确认。 *)
    bLimitsValid : BOOL;
    (* 标准NC Adapter报告轴已使能且可接管。 *)
    bAxisReady : BOOL;
    (* 标准NC Adapter或轴报告错误。 *)
    bAxisError : BOOL;
    (* 实际Fast/SAF同步周期，单位秒。 *)
    rCycleTime_s : LREAL;
    (* Z轴最小允许位置，单位毫米。 *)
    rMinimumPosition_mm : LREAL;
    (* Z轴最大允许位置，单位毫米。 *)
    rMaximumPosition_mm : LREAL;
    (* Z轴绝对最大速度，单位毫米每秒。 *)
    rMaximumVelocity_mm_s : LREAL;
    (* Z轴绝对最大加速度，单位毫米每二次方秒。 *)
    rMaximumAcceleration_mm_s2 : LREAL;
    (* External Setpoint受控配置。 *)
    stConfig : ST_ZExtSetpointConfig;
    (* Enable/Feed/Disable及P/V/A/Direction命令。 *)
    stCommand : ST_ZExtSetpointCommand;
END_VAR
VAR_OUTPUT
    (* External Setpoint生命周期状态。 *)
    stStatus : ST_ZExtSetpointStatus;
END_VAR
VAR
    (* NC External Setpoint使能实例。 *)
    fbEnable : MC_ExtSetPointGenEnable;
    (* NC External Setpoint禁用实例。 *)
    fbDisable : MC_ExtSetPointGenDisable;
    (* 等待使能确认超时实例。 *)
    fbEnableTimeout : TON;
    (* 等待禁用确认超时实例。 *)
    fbDisableTimeout : TON;
    (* 当前生命周期状态。 *)
    eState : E_ZExtSetpointState;
    (* 当前扫描使能Execute脉冲。 *)
    bEnablePulse : BOOL;
    (* 当前扫描禁用Execute脉冲。 *)
    bDisablePulse : BOOL;
    (* 当前扫描必须写入P/V/A/Direction。 *)
    bFeedThisCycle : BOOL;
    (* MC_ExtSetPointGenFeed未使用的函数返回值。 *)
    bFeedUnused : BOOL;
    (* Enable前真实NC初值、轴健康、Owner、配置和限值检查结果。 *)
    bPrecheckOk : BOOL;
    (* Active期当前Feed包通过有限值、边界和方向基本检查。 *)
    bActiveFeedCommandValid : BOOL;
    (* 当前命令与上一Feed满足连续性窗口。 *)
    bContinuityValid : BOOL;
    (* 当前送入NC的外部位置，单位毫米。 *)
    rFeedPosition_mm : LREAL;
    (* 当前送入NC的外部速度，单位毫米每秒。 *)
    rFeedVelocity_mm_s : LREAL;
    (* 当前送入NC的外部加速度，单位毫米每二次方秒。 *)
    rFeedAcceleration_mm_s2 : LREAL;
    (* 当前送入NC的方向，只允许-1、0、1。 *)
    nFeedDirection : DINT;
    (* Precheck从真实NC速度推导的初始方向。 *)
    nInitialDirection : DINT;
    (* 退出前最后一个非零方向。 *)
    nLastNonZeroDirection : DINT;
    (* Active内换向已接受旧方向静止包。 *)
    bZ_EXT_DIRECTION_HOLD : BOOL;
    (* Active内换向已接受Direction=0静止包。 *)
    bZ_EXT_DIRECTION_ZERO : BOOL;
    (* Active内换向已接受新非零Direction静止预置包。 *)
    bZ_EXT_DIRECTION_PRELOAD : BOOL;
    (* 已预置但尚未开始运动的新方向。 *)
    nPendingDirection : DINT;
    (* 本扫描Feed前的accepted方向快照。 *)
    nAcceptedDirection : DINT;
    (* 硬正向抑制包已在本扫描接受，下一扫描消费Disable。 *)
    bDisable : BOOL;
    (* 本扫描普通非静止Feed接受后清除方向握手状态。 *)
    bClearDirectionHandshakeAfterFeed : BOOL;
    (* 梯形积分使用的上周期速度。 *)
    rPreviousVelocity_mm_s : LREAL;
    (* 连续性检查的期望位置。 *)
    rExpectedPosition_mm : LREAL;
    (* 当前状态内扫描计数。 *)
    nStateCycleCounter : UINT;
    (* Feed总扫描计数。 *)
    udiFeedCycleCounter : UDINT;
    (* 生命周期错误锁存编号。 *)
    udiLatchedErrorId : UDINT;
    (* 本扫描Active Feed安全检查的故障候选，非零时同扫描锁存。 *)
    nFaultId : UDINT;
    (* 完整退出结束后应进入ERROR而不是DONE。 *)
    bExitDueToError : BOOL;
    (* 已进入Disable阶段，释放Owner前必须完成Disabled确认和后保持。 *)
    bPostDisableHoldPending : BOOL;
END_VAR

(* ---------------------------------------------------------
   Z轴External Setpoint生命周期状态机。
   进入：标准NC已使能、Owner已授予、真实驱动已绑定、配置和限值有效。
   动作：预置NC当前SetPos/SetVelo/SetAcc，Enable后每SAF Feed。
   成功：速度归零、保持Direction、Direction清零、Disable并后保持。
   超时：Enable/Disable超时锁存ALARM_EXTERNAL_SETPOINT_FAULT来源。
   Fault：先尝试完整退出；未确认Disabled前绝不释放Owner。
   --------------------------------------------------------- *)
bEnablePulse := FALSE;
bDisablePulse := FALSE;
bFeedThisCycle := FALSE;
bClearDirectionHandshakeAfterFeed := FALSE;
stStatus.bFeedAccepted := FALSE;
nAcceptedDirection := stStatus.nAcceptedDirection;
nFaultId := 0;

(* Enable前只检查真实NC初值与生命周期条件，不要求上层尚未生成的Feed包。 *)
bPrecheckOk := stConfig.bValid
    AND bDriveLinked AND bOwnerGranted AND bLimitsValid
    AND bAxisReady AND NOT bAxisError
    AND (rCycleTime_s > 0.0)
    AND FC_IsFiniteLReal(rValue := rCycleTime_s)
    AND (stConfig.tEnableTimeout > T#0S)
    AND (stConfig.tDisableTimeout > T#0S)
    AND FC_IsFiniteLReal(rValue := rMinimumPosition_mm)
    AND FC_IsFiniteLReal(rValue := rMaximumPosition_mm)
    AND FC_IsFiniteLReal(rValue := rMaximumVelocity_mm_s)
    AND FC_IsFiniteLReal(rValue := rMaximumAcceleration_mm_s2)
    AND (rMaximumPosition_mm > rMinimumPosition_mm)
    AND (ABS(rMaximumVelocity_mm_s) > 0.0)
    AND (ABS(rMaximumAcceleration_mm_s2) > 0.0)
    AND FC_IsFiniteLReal(rValue := stConfig.rStandstillVelocity_mm_s)
    AND FC_IsFiniteLReal(rValue := stConfig.rMaximumPositionDeviation_mm)
    AND FC_IsFiniteLReal(rValue := stConfig.rMaximumVelocityStep_mm_s)
    AND FC_IsFiniteLReal(rValue := Axis.NcToPlc.SetPos)
    AND FC_IsFiniteLReal(rValue := Axis.NcToPlc.SetVelo)
    AND FC_IsFiniteLReal(rValue := Axis.NcToPlc.SetAcc)
    AND (Axis.NcToPlc.SetPos >= rMinimumPosition_mm)
    AND (Axis.NcToPlc.SetPos <= rMaximumPosition_mm)
    AND (ABS(Axis.NcToPlc.SetVelo) <= ABS(rMaximumVelocity_mm_s))
    AND (ABS(Axis.NcToPlc.SetAcc) <= ABS(rMaximumAcceleration_mm_s2))
    AND (stConfig.rStandstillVelocity_mm_s >= 0.0)
    AND (stConfig.rMaximumPositionDeviation_mm >= 0.0)
    AND (stConfig.rMaximumVelocityStep_mm_s >= 0.0)
    AND (stConfig.nDirectionHoldCycles >= 1)
    AND (stConfig.nPostDisableHoldCycles >= 1);

(* Active Feed额外检查命令本身；连续性和换向握手在ACTIVE分支中检查。 *)
bActiveFeedCommandValid := bPrecheckOk
    AND FC_IsFiniteLReal(rValue := stCommand.rPosition_mm)
    AND FC_IsFiniteLReal(rValue := stCommand.rVelocity_mm_s)
    AND FC_IsFiniteLReal(rValue := stCommand.rAcceleration_mm_s2)
    AND (stCommand.nDirection >= -1) AND (stCommand.nDirection <= 1)
    AND (stCommand.rPosition_mm >= rMinimumPosition_mm)
    AND (stCommand.rPosition_mm <= rMaximumPosition_mm)
    AND (ABS(stCommand.rVelocity_mm_s) <= ABS(rMaximumVelocity_mm_s))
    AND (ABS(stCommand.rAcceleration_mm_s2) <= ABS(rMaximumAcceleration_mm_s2));

IF stCommand.rVelocity_mm_s > stConfig.rStandstillVelocity_mm_s THEN
    bActiveFeedCommandValid := bActiveFeedCommandValid AND (stCommand.nDirection = 1);
ELSIF stCommand.rVelocity_mm_s < -stConfig.rStandstillVelocity_mm_s THEN
    bActiveFeedCommandValid := bActiveFeedCommandValid AND (stCommand.nDirection = -1);
END_IF

fbEnableTimeout(
    IN := eState = E_ZExtSetpointState.Z_EXT_WAIT_ENABLED,
    PT := stConfig.tEnableTimeout);
fbDisableTimeout(
    IN := eState = E_ZExtSetpointState.Z_EXT_WAIT_DISABLED,
    PT := stConfig.tDisableTimeout);

CASE eState OF
    E_ZExtSetpointState.Z_EXT_IDLE:
        stStatus.bDone := FALSE;
        stStatus.bReleaseOwner := FALSE;
        stStatus.bAcceptedSetpointValid := FALSE;
        nStateCycleCounter := 0;
        bZ_EXT_DIRECTION_HOLD := FALSE;
        bZ_EXT_DIRECTION_ZERO := FALSE;
        bZ_EXT_DIRECTION_PRELOAD := FALSE;
        nPendingDirection := 0;
        bDisable := FALSE;
        IF stCommand.bReset THEN
            udiLatchedErrorId := 0;
            bExitDueToError := FALSE;
        END_IF
        IF stCommand.bEnable AND bOwnerGranted THEN
            eState := E_ZExtSetpointState.Z_EXT_PRECHECK;
        END_IF

    E_ZExtSetpointState.Z_EXT_PRECHECK:
        (* 每次新Precheck先清除有效标志，不伪造accepted数值。 *)
        stStatus.bAcceptedSetpointValid := FALSE;
        IF NOT bOwnerGranted THEN
            udiLatchedErrorId := 16#00007202;
            bExitDueToError := TRUE;
            eState := E_ZExtSetpointState.Z_EXT_ERROR;
        ELSIF NOT bPrecheckOk THEN
            udiLatchedErrorId := 16#00007201;
            bExitDueToError := TRUE;
            eState := E_ZExtSetpointState.Z_EXT_ERROR;
        ELSE
            (* 从本机Tc2_MC2实际NCTOPLC字段取得无扰接管初值。 *)
            rFeedPosition_mm := Axis.NcToPlc.SetPos;
            rFeedVelocity_mm_s := Axis.NcToPlc.SetVelo;
            rFeedAcceleration_mm_s2 := Axis.NcToPlc.SetAcc;
            nInitialDirection := 0;
            IF rFeedVelocity_mm_s > stConfig.rStandstillVelocity_mm_s THEN
                nInitialDirection := 1;
            ELSIF rFeedVelocity_mm_s < -stConfig.rStandstillVelocity_mm_s THEN
                nInitialDirection := -1;
            END_IF
            nFeedDirection := nInitialDirection;
            (* 新生命周期不得继承上一周期的非零方向。 *)
            nLastNonZeroDirection := nInitialDirection;
            rPreviousVelocity_mm_s := rFeedVelocity_mm_s;
            bZ_EXT_DIRECTION_HOLD := FALSE;
            bZ_EXT_DIRECTION_ZERO := FALSE;
            bZ_EXT_DIRECTION_PRELOAD := FALSE;
            nPendingDirection := 0;
            bDisable := FALSE;
            stStatus.bAcceptedSetpointValid := TRUE;
            stStatus.rAcceptedPosition_mm := Axis.NcToPlc.SetPos;
            stStatus.rAcceptedVelocity_mm_s := Axis.NcToPlc.SetVelo;
            stStatus.rAcceptedAcceleration_mm_s2 := Axis.NcToPlc.SetAcc;
            stStatus.nAcceptedDirection := nInitialDirection;
            eState := E_ZExtSetpointState.Z_EXT_PRELOAD_DIRECTION;
        END_IF

    E_ZExtSetpointState.Z_EXT_PRELOAD_DIRECTION:
        bFeedThisCycle := TRUE;
        eState := E_ZExtSetpointState.Z_EXT_PREFEED_INITIAL;

    E_ZExtSetpointState.Z_EXT_PREFEED_INITIAL:
        bFeedThisCycle := TRUE;
        eState := E_ZExtSetpointState.Z_EXT_ENABLE;

    E_ZExtSetpointState.Z_EXT_ENABLE:
        bFeedThisCycle := TRUE;
        IF NOT bOwnerGranted THEN
            udiLatchedErrorId := 16#00007202;
            bExitDueToError := TRUE;
            eState := E_ZExtSetpointState.Z_EXT_RAMP_TO_ZERO;
        ELSIF NOT bPrecheckOk THEN
            udiLatchedErrorId := 16#00007201;
            bExitDueToError := TRUE;
            eState := E_ZExtSetpointState.Z_EXT_RAMP_TO_ZERO;
        ELSE
            bEnablePulse := bOwnerGranted AND bDriveLinked AND bAxisReady;
            eState := E_ZExtSetpointState.Z_EXT_WAIT_ENABLED;
        END_IF

    E_ZExtSetpointState.Z_EXT_WAIT_ENABLED:
        bFeedThisCycle := TRUE;
        IF fbEnable.Error THEN
            bFeedThisCycle := FALSE;
            udiLatchedErrorId := fbEnable.ErrorID;
            bExitDueToError := TRUE;
            eState := E_ZExtSetpointState.Z_EXT_RAMP_TO_ZERO;
        ELSIF NOT bOwnerGranted THEN
            bFeedThisCycle := FALSE;
            udiLatchedErrorId := 16#00007202;
            bExitDueToError := TRUE;
            eState := E_ZExtSetpointState.Z_EXT_RAMP_TO_ZERO;
        ELSIF NOT bPrecheckOk THEN
            (* Enable确认前健康、配置或真实NC初值失效时禁止本扫描Feed。 *)
            bFeedThisCycle := FALSE;
            udiLatchedErrorId := 16#00007201;
            bExitDueToError := TRUE;
            eState := E_ZExtSetpointState.Z_EXT_RAMP_TO_ZERO;
        ELSIF Axis.Status.ExtSetPointGenEnabled OR fbEnable.Enabled THEN
            IF stCommand.bPositiveMotionInhibit THEN
                (* Enable确认扫描也必须在MC Feed前完成硬抑制包校验。 *)
                IF stCommand.bFeed
                    AND bActiveFeedCommandValid
                    AND stStatus.bAcceptedSetpointValid
                    AND (stCommand.rPosition_mm = stStatus.rAcceptedPosition_mm)
                    AND (stCommand.rVelocity_mm_s = 0.0)
                    AND (stCommand.rAcceleration_mm_s2 = 0.0)
                    AND (stCommand.nDirection = stStatus.nAcceptedDirection) THEN
                    rFeedPosition_mm := stStatus.rAcceptedPosition_mm;
                    rFeedVelocity_mm_s := 0.0;
                    rFeedAcceleration_mm_s2 := 0.0;
                    nFeedDirection := stStatus.nAcceptedDirection;
                    bFeedThisCycle := TRUE;
                    bDisable := TRUE;
                    rPreviousVelocity_mm_s := rFeedVelocity_mm_s;
                    eState := E_ZExtSetpointState.Z_EXT_ACTIVE;
                ELSE
                    bFeedThisCycle := FALSE;
                    udiLatchedErrorId := 16#0000720A;
                    bExitDueToError := TRUE;
                    eState := E_ZExtSetpointState.Z_EXT_RAMP_TO_ZERO;
                END_IF
            ELSE
                rPreviousVelocity_mm_s := rFeedVelocity_mm_s;
                eState := E_ZExtSetpointState.Z_EXT_ACTIVE;
            END_IF
        ELSIF fbEnableTimeout.Q THEN
            bFeedThisCycle := FALSE;
            udiLatchedErrorId := 16#00007204;
            bExitDueToError := TRUE;
            eState := E_ZExtSetpointState.Z_EXT_RAMP_TO_ZERO;
        END_IF

    E_ZExtSetpointState.Z_EXT_ACTIVE:
        (* 固定优先级：轴/Owner健康 -> 已接受硬抑制的Disable -> 硬抑制包 ->
           普通Disable/Reset -> 普通Feed与Active内双阶段换向。 *)
        IF NOT bDriveLinked OR NOT bOwnerGranted OR NOT bAxisReady OR bAxisError THEN
            IF NOT bOwnerGranted THEN
                udiLatchedErrorId := 16#00007202;
            ELSE
                udiLatchedErrorId := 16#00007201;
            END_IF
            bExitDueToError := TRUE;
            eState := E_ZExtSetpointState.Z_EXT_RAMP_TO_ZERO;
        ELSIF bDisable THEN
            (* 硬抑制零速包已在上一扫描接受，本扫描进入既有完整Disable序列。 *)
            bDisable := FALSE;
            eState := E_ZExtSetpointState.Z_EXT_RAMP_TO_ZERO;
        ELSIF stCommand.bPositiveMotionInhibit THEN
            (* 唯一允许绕过Velocity-Step的包：保持accepted P/方向，V/A立即为零。 *)
            IF stCommand.bFeed
                AND bActiveFeedCommandValid
                AND stStatus.bAcceptedSetpointValid
                AND (stCommand.rPosition_mm = stStatus.rAcceptedPosition_mm)
                AND (stCommand.rVelocity_mm_s = 0.0)
                AND (stCommand.rAcceleration_mm_s2 = 0.0)
                AND (stCommand.nDirection = stStatus.nAcceptedDirection) THEN
                rFeedPosition_mm := stStatus.rAcceptedPosition_mm;
                rFeedVelocity_mm_s := 0.0;
                rFeedAcceleration_mm_s2 := 0.0;
                nFeedDirection := stStatus.nAcceptedDirection;
                bFeedThisCycle := TRUE;
                (* 只接受一包；下一扫描由内部Disable请求进入安全退出。 *)
                bDisable := TRUE;
            ELSE
                udiLatchedErrorId := 16#0000720A;
                bExitDueToError := TRUE;
                eState := E_ZExtSetpointState.Z_EXT_RAMP_TO_ZERO;
            END_IF
        ELSIF stCommand.bDisable OR stCommand.bReset OR NOT stCommand.bEnable THEN
            eState := E_ZExtSetpointState.Z_EXT_RAMP_TO_ZERO;
        ELSIF NOT stCommand.bFeed OR NOT bActiveFeedCommandValid THEN
            udiLatchedErrorId := 16#00007207;
            bExitDueToError := TRUE;
            eState := E_ZExtSetpointState.Z_EXT_RAMP_TO_ZERO;
        ELSE
            nFeedDirection := stCommand.nDirection;

            IF ((nAcceptedDirection = 1) AND (nFeedDirection = -1))
                OR ((nAcceptedDirection = -1) AND (nFeedDirection = 1)) THEN
                (* +1/-1不得直接跳变。 *)
                nFaultId := 16#00007209;
                udiLatchedErrorId := nFaultId;
                bExitDueToError := TRUE;
                eState := E_ZExtSetpointState.Z_EXT_RAMP_TO_ZERO;
            ELSIF (nFeedDirection <> stStatus.nAcceptedDirection)
                AND ((stCommand.rVelocity_mm_s <> 0.0)
                    OR (stCommand.rAcceleration_mm_s2 <> 0.0)
                    OR (stCommand.rPosition_mm <> stStatus.rAcceptedPosition_mm)) THEN
                (* 任何方向变化都必须使用held-P/V0/A0静止包。 *)
                udiLatchedErrorId := 16#00007209;
                bExitDueToError := TRUE;
                eState := E_ZExtSetpointState.Z_EXT_RAMP_TO_ZERO;
            ELSIF (nFeedDirection = stStatus.nAcceptedDirection)
                AND (nFeedDirection <> 0)
                AND (stStatus.rAcceptedVelocity_mm_s = 0.0)
                AND (stCommand.rVelocity_mm_s = 0.0)
                AND (stCommand.rAcceleration_mm_s2 = 0.0)
                AND (stCommand.rPosition_mm <> stStatus.rAcceptedPosition_mm) THEN
                (* 旧方向已静止时也必须严格held accepted-P，禁止窗口内位置偷跳。 *)
                udiLatchedErrorId := 16#00007209;
                bExitDueToError := TRUE;
                eState := E_ZExtSetpointState.Z_EXT_RAMP_TO_ZERO;
            ELSIF (nFeedDirection = stStatus.nAcceptedDirection)
                AND (nFeedDirection <> 0)
                AND (stStatus.rAcceptedVelocity_mm_s = 0.0)
                AND (stCommand.rPosition_mm = stStatus.rAcceptedPosition_mm)
                AND (stCommand.rVelocity_mm_s = 0.0)
                AND (stCommand.rAcceleration_mm_s2 = 0.0) THEN
                (* 旧方向静止Feed是换向的第一接受阶段。 *)
                bZ_EXT_DIRECTION_HOLD := TRUE;
                rFeedPosition_mm := stCommand.rPosition_mm;
                rFeedVelocity_mm_s := 0.0;
                rFeedAcceleration_mm_s2 := 0.0;
                bFeedThisCycle := TRUE;
            ELSIF (nFeedDirection = 0)
                AND (stStatus.nAcceptedDirection <> 0) THEN
                IF NOT bZ_EXT_DIRECTION_HOLD THEN
                    udiLatchedErrorId := 16#00007209;
                    bExitDueToError := TRUE;
                    eState := E_ZExtSetpointState.Z_EXT_RAMP_TO_ZERO;
                ELSE
                    (* 第二阶段：保持位置并接受Direction=0一个完整周期。 *)
                    bZ_EXT_DIRECTION_ZERO := TRUE;
                    bZ_EXT_DIRECTION_PRELOAD := FALSE;
                    nPendingDirection := 0;
                    rFeedPosition_mm := stStatus.rAcceptedPosition_mm;
                    rFeedVelocity_mm_s := 0.0;
                    rFeedAcceleration_mm_s2 := 0.0;
                    bFeedThisCycle := TRUE;
                END_IF
            ELSIF (stStatus.nAcceptedDirection = 0)
                AND (nFeedDirection <> 0) THEN
                IF NOT bZ_EXT_DIRECTION_ZERO THEN
                    udiLatchedErrorId := 16#00007209;
                    bExitDueToError := TRUE;
                    eState := E_ZExtSetpointState.Z_EXT_RAMP_TO_ZERO;
                ELSE
                    (* 第三阶段：新非零方向必须先接受一个held-P/V0/A0预置包。 *)
                    nPendingDirection := nFeedDirection;
                    bZ_EXT_DIRECTION_PRELOAD := TRUE;
                    rFeedPosition_mm := stStatus.rAcceptedPosition_mm;
                    rFeedVelocity_mm_s := 0.0;
                    rFeedAcceleration_mm_s2 := 0.0;
                    bFeedThisCycle := TRUE;
                END_IF
            ELSIF (nFeedDirection = 0)
                AND ((stCommand.rPosition_mm <> stStatus.rAcceptedPosition_mm)
                    OR (stCommand.rVelocity_mm_s <> 0.0)
                    OR (stCommand.rAcceleration_mm_s2 <> 0.0)) THEN
                udiLatchedErrorId := 16#00007209;
                bExitDueToError := TRUE;
                eState := E_ZExtSetpointState.Z_EXT_RAMP_TO_ZERO;
            ELSIF (bZ_EXT_DIRECTION_PRELOAD)
                AND ((nFeedDirection <> nPendingDirection)
                    OR (stStatus.nAcceptedDirection <> nPendingDirection)) THEN
                (* 新方向移动必须晚于一个已接受的新方向预置包。 *)
                udiLatchedErrorId := 16#00007209;
                bExitDueToError := TRUE;
                eState := E_ZExtSetpointState.Z_EXT_RAMP_TO_ZERO;
            ELSE
                rExpectedPosition_mm := stStatus.rAcceptedPosition_mm
                    + 0.5 * (stStatus.rAcceptedVelocity_mm_s + stCommand.rVelocity_mm_s)
                    * rCycleTime_s;
                bContinuityValid := ABS(stCommand.rPosition_mm - rExpectedPosition_mm)
                        <= stConfig.rMaximumPositionDeviation_mm
                    AND ABS(stCommand.rVelocity_mm_s - stStatus.rAcceptedVelocity_mm_s)
                        <= stConfig.rMaximumVelocityStep_mm_s;
                IF NOT bContinuityValid THEN
                    udiLatchedErrorId := 16#00007208;
                    bExitDueToError := TRUE;
                    eState := E_ZExtSetpointState.Z_EXT_RAMP_TO_ZERO;
                ELSE
                    rFeedPosition_mm := stCommand.rPosition_mm;
                    rFeedVelocity_mm_s := stCommand.rVelocity_mm_s;
                    rFeedAcceleration_mm_s2 := stCommand.rAcceleration_mm_s2;
                    IF nFeedDirection <> 0 THEN
                        nLastNonZeroDirection := nFeedDirection;
                    END_IF
                    rPreviousVelocity_mm_s := rFeedVelocity_mm_s;
                    bFeedThisCycle := TRUE;
                    IF (stCommand.rPosition_mm <> stStatus.rAcceptedPosition_mm)
                        OR (stCommand.rVelocity_mm_s <> 0.0)
                        OR (stCommand.rAcceleration_mm_s2 <> 0.0) THEN
                        bClearDirectionHandshakeAfterFeed := TRUE;
                    END_IF
                END_IF
            END_IF
        END_IF

    E_ZExtSetpointState.Z_EXT_RAMP_TO_ZERO:
        IF rCycleTime_s > 0.0 THEN
            rPreviousVelocity_mm_s := rFeedVelocity_mm_s;
            rFeedVelocity_mm_s := FC_LimitRate(
                rCurrent := rFeedVelocity_mm_s,
                rTarget := 0.0,
                rRateUpPer_s := ABS(rMaximumAcceleration_mm_s2),
                rRateDownPer_s := ABS(rMaximumAcceleration_mm_s2),
                rCycleTime_s := rCycleTime_s);
            rFeedAcceleration_mm_s2 := (rFeedVelocity_mm_s - rPreviousVelocity_mm_s) / rCycleTime_s;
            rFeedPosition_mm := rFeedPosition_mm
                + 0.5 * (rPreviousVelocity_mm_s + rFeedVelocity_mm_s) * rCycleTime_s;
        ELSE
            rFeedVelocity_mm_s := 0.0;
            rFeedAcceleration_mm_s2 := 0.0;
        END_IF
        IF rFeedVelocity_mm_s > stConfig.rStandstillVelocity_mm_s THEN
            nLastNonZeroDirection := 1;
        ELSIF rFeedVelocity_mm_s < -stConfig.rStandstillVelocity_mm_s THEN
            nLastNonZeroDirection := -1;
        END_IF
        nFeedDirection := nLastNonZeroDirection;
        bFeedThisCycle := bDriveLinked;
        IF ABS(rFeedVelocity_mm_s) <= stConfig.rStandstillVelocity_mm_s THEN
            rFeedVelocity_mm_s := 0.0;
            rFeedAcceleration_mm_s2 := 0.0;
            nStateCycleCounter := 0;
            eState := E_ZExtSetpointState.Z_EXT_HOLD_DIRECTION;
        END_IF

    E_ZExtSetpointState.Z_EXT_HOLD_DIRECTION:
        rFeedVelocity_mm_s := 0.0;
        rFeedAcceleration_mm_s2 := 0.0;
        nFeedDirection := nLastNonZeroDirection;
        bFeedThisCycle := bDriveLinked;
        nStateCycleCounter := nStateCycleCounter + 1;
        IF nStateCycleCounter >= stConfig.nDirectionHoldCycles THEN
            nStateCycleCounter := 0;
            eState := E_ZExtSetpointState.Z_EXT_DIRECTION_ZERO;
        END_IF

    E_ZExtSetpointState.Z_EXT_DIRECTION_ZERO:
        rFeedVelocity_mm_s := 0.0;
        rFeedAcceleration_mm_s2 := 0.0;
        nFeedDirection := 0;
        bFeedThisCycle := bDriveLinked;
        eState := E_ZExtSetpointState.Z_EXT_DISABLE;

    E_ZExtSetpointState.Z_EXT_DISABLE:
        bFeedThisCycle := bDriveLinked;
        bDisablePulse := bDriveLinked;
        bPostDisableHoldPending := TRUE;
        nStateCycleCounter := 0;
        eState := E_ZExtSetpointState.Z_EXT_WAIT_DISABLED;

    E_ZExtSetpointState.Z_EXT_WAIT_DISABLED:
        (* Beckhoff规定Disable后外部目标还会再接收一个周期。 *)
        bFeedThisCycle := bDriveLinked;
        nStateCycleCounter := nStateCycleCounter + 1;
        IF fbDisable.Error THEN
            udiLatchedErrorId := fbDisable.ErrorID;
            bExitDueToError := TRUE;
            eState := E_ZExtSetpointState.Z_EXT_ERROR;
        ELSIF NOT Axis.Status.ExtSetPointGenEnabled
            AND NOT fbEnable.Enabled AND NOT fbDisable.Enabled
            AND (nStateCycleCounter >= 1) THEN
            nStateCycleCounter := 0;
            eState := E_ZExtSetpointState.Z_EXT_POST_DISABLE_HOLD;
        ELSIF fbDisableTimeout.Q THEN
            udiLatchedErrorId := 16#00007205;
            bExitDueToError := TRUE;
            eState := E_ZExtSetpointState.Z_EXT_ERROR;
        END_IF

    E_ZExtSetpointState.Z_EXT_POST_DISABLE_HOLD:
        bFeedThisCycle := bDriveLinked;
        nStateCycleCounter := nStateCycleCounter + 1;
        IF nStateCycleCounter >= stConfig.nPostDisableHoldCycles THEN
            bPostDisableHoldPending := FALSE;
            IF bExitDueToError THEN
                eState := E_ZExtSetpointState.Z_EXT_ERROR;
            ELSE
                eState := E_ZExtSetpointState.Z_EXT_DONE;
            END_IF
        END_IF

    E_ZExtSetpointState.Z_EXT_DONE:
        stStatus.bDone := TRUE;
        stStatus.bReleaseOwner := TRUE;
        IF NOT stCommand.bEnable THEN
            stStatus.bAcceptedSetpointValid := FALSE;
            bZ_EXT_DIRECTION_HOLD := FALSE;
            bZ_EXT_DIRECTION_ZERO := FALSE;
            bZ_EXT_DIRECTION_PRELOAD := FALSE;
            nPendingDirection := 0;
            bDisable := FALSE;
            eState := E_ZExtSetpointState.Z_EXT_IDLE;
        END_IF

    E_ZExtSetpointState.Z_EXT_ERROR:
        stStatus.bDone := FALSE;
        bFeedThisCycle := bPostDisableHoldPending AND bDriveLinked;
        stStatus.bReleaseOwner := NOT bPostDisableHoldPending AND NOT Axis.Status.ExtSetPointGenEnabled
            AND NOT fbEnable.Enabled AND NOT fbDisable.Enabled;
        IF bPostDisableHoldPending AND NOT Axis.Status.ExtSetPointGenEnabled
            AND NOT fbEnable.Enabled AND NOT fbDisable.Enabled THEN
            nStateCycleCounter := 0;
            eState := E_ZExtSetpointState.Z_EXT_POST_DISABLE_HOLD;
        ELSIF bPostDisableHoldPending AND stCommand.bReset AND bDriveLinked THEN
            eState := E_ZExtSetpointState.Z_EXT_DISABLE;
        ELSIF stCommand.bReset AND NOT stCommand.bEnable AND stStatus.bReleaseOwner THEN
            udiLatchedErrorId := 0;
            bExitDueToError := FALSE;
            stStatus.bAcceptedSetpointValid := FALSE;
            bZ_EXT_DIRECTION_HOLD := FALSE;
            bZ_EXT_DIRECTION_ZERO := FALSE;
            bZ_EXT_DIRECTION_PRELOAD := FALSE;
            nPendingDirection := 0;
            bDisable := FALSE;
            eState := E_ZExtSetpointState.Z_EXT_IDLE;
        END_IF

    ELSE
        udiLatchedErrorId := 16#00007206;
        bExitDueToError := TRUE;
        stStatus.bDone := FALSE;
        stStatus.bReleaseOwner := FALSE;
        stStatus.bAcceptedSetpointValid := FALSE;
        bFeedThisCycle := FALSE;
        IF Axis.Status.ExtSetPointGenEnabled OR fbEnable.Enabled OR fbDisable.Enabled THEN
            bPostDisableHoldPending := TRUE;
            eState := E_ZExtSetpointState.Z_EXT_DISABLE;
        ELSE
            bPostDisableHoldPending := FALSE;
            eState := E_ZExtSetpointState.Z_EXT_ERROR;
        END_IF
END_CASE

fbEnable(
    Axis := Axis,
    Execute := bEnablePulse,
    Position := rFeedPosition_mm,
    PositionType := POSITIONTYPE_ABSOLUTE);
fbDisable(Axis := Axis, Execute := bDisablePulse);

IF bFeedThisCycle AND bDriveLinked THEN
    bFeedUnused := MC_ExtSetPointGenFeed(
        Axis := Axis,
        Position := rFeedPosition_mm,
        Velocity := rFeedVelocity_mm_s,
        Acceleration := rFeedAcceleration_mm_s2,
        Direction := nFeedDirection);
    IF udiFeedCycleCounter = UDINT#4294967295 THEN
        udiFeedCycleCounter := 1;
    ELSE
        udiFeedCycleCounter := udiFeedCycleCounter + 1;
    END_IF
    (* 所有安全检查已在MC Feed前完成；这是唯一accepted发布点。 *)
    stStatus.bFeedAccepted := TRUE;
    stStatus.bAcceptedSetpointValid := TRUE;
    stStatus.rAcceptedPosition_mm := rFeedPosition_mm;
    stStatus.rAcceptedVelocity_mm_s := rFeedVelocity_mm_s;
    stStatus.rAcceptedAcceleration_mm_s2 := rFeedAcceleration_mm_s2;
    stStatus.nAcceptedDirection := nFeedDirection;

    IF bClearDirectionHandshakeAfterFeed THEN
        bZ_EXT_DIRECTION_HOLD := FALSE;
        bZ_EXT_DIRECTION_ZERO := FALSE;
        bZ_EXT_DIRECTION_PRELOAD := FALSE;
        nPendingDirection := 0;
    END_IF

    (* 初始静止Feed也是真实accepted Direction=0阶段，可安全启动新方向预置。 *)
    IF (nFeedDirection = 0)
        AND (ABS(rFeedVelocity_mm_s) <= stConfig.rStandstillVelocity_mm_s)
        AND (rFeedAcceleration_mm_s2 = 0.0) THEN
        bZ_EXT_DIRECTION_ZERO := TRUE;
        bZ_EXT_DIRECTION_PRELOAD := FALSE;
        nPendingDirection := 0;
    ELSIF bZ_EXT_DIRECTION_ZERO
        AND (nFeedDirection <> 0)
        AND (ABS(rFeedVelocity_mm_s) <= stConfig.rStandstillVelocity_mm_s)
        AND (rFeedAcceleration_mm_s2 = 0.0) THEN
        nPendingDirection := nFeedDirection;
        bZ_EXT_DIRECTION_PRELOAD := TRUE;
    END_IF
END_IF

stStatus.eState := eState;
stStatus.bEnabled := bDriveLinked AND (Axis.Status.ExtSetPointGenEnabled
    OR fbEnable.Enabled OR fbDisable.Enabled);
stStatus.bBusy := (eState <> E_ZExtSetpointState.Z_EXT_IDLE)
    AND (eState <> E_ZExtSetpointState.Z_EXT_DONE)
    AND (eState <> E_ZExtSetpointState.Z_EXT_ERROR);
stStatus.bError := udiLatchedErrorId <> 0;
stStatus.nErrorId := udiLatchedErrorId;
stStatus.udiFeedCycleCounter := udiFeedCycleCounter;

END_FUNCTION_BLOCK

// ---- POUs/FunctionBlocks/Axis/FB_RAxisNcAdapter.TcPOU
FUNCTION_BLOCK FB_RAxisNcAdapter
VAR_IN_OUT
    (* 唯一R轴NC引用；仅允许本Adapter访问。 *)
    Axis : AXIS_REF;
END_VAR
VAR_INPUT
    (* 真实驱动、编码器和NC轴已经人工关联并验证。 *)
    bDriveLinked : BOOL;
    (* 上层命令事务编号；只有变化才产生MC Execute上升沿。 *)
    udiCommandId : UDINT;
    (* R轴标准RPM命令；首版不包含扭矩闭环。 *)
    stCommand : ST_RAxisCommand;
END_VAR
VAR_OUTPUT
    (* R轴标准运动状态快照。 *)
    stStatus : ST_RAxisStatus;
    (* Adapter已处理的最后命令事务编号。 *)
    udiAcceptedCommandId : UDINT;
END_VAR
VAR
    (* R轴软件使能实例。 *)
    fbPower : MC_Power;
    (* R轴错误复位实例。 *)
    fbReset : MC_Reset;
    (* R轴速度运动双实例A，用于替换活动速度命令。 *)
    fbMoveVelocityA : MC_MoveVelocity;
    (* R轴速度运动双实例B，用于替换活动速度命令。 *)
    fbMoveVelocityB : MC_MoveVelocity;
    (* R轴受控停止实例。 *)
    fbHalt : MC_Halt;
    (* 当前扫描检测到新的命令编号。 *)
    bNewCommand : BOOL;
    (* 当前扫描的复位Execute脉冲。 *)
    bResetPulse : BOOL;
    (* 当前扫描速度实例A的Execute脉冲。 *)
    bMoveVelocityPulseA : BOOL;
    (* 当前扫描速度实例B的Execute脉冲。 *)
    bMoveVelocityPulseB : BOOL;
    (* 当前扫描的受控停止Execute脉冲。 *)
    bHaltPulse : BOOL;
    (* 下次速度命令选择A实例，否则选择B实例。 *)
    bSelectVelocityA : BOOL;
    (* RPM命令方向。 *)
    eVelocityDirection : MC_Direction;
END_VAR

(* ---------------------------------------------------------
   R轴标准NC Adapter状态。
   进入：Task_CffFast每扫描调用，且由PRG_FastAxisControl唯一持有。
   动作：更新AXIS_REF状态；命令编号变化时产生一次RPM命令上升沿。
   成功：发布RPM与只读Torque；Ready要求真实驱动人工关联。
   超时：由上层流程负责；MC Busy/Error保持可诊断。
   Fault：Stop优先；未绑定驱动时Power和全部运动Execute硬门控。
   --------------------------------------------------------- *)
Axis.ReadStatus();

bNewCommand := udiCommandId <> udiAcceptedCommandId;
bResetPulse := FALSE;
bMoveVelocityPulseA := FALSE;
bMoveVelocityPulseB := FALSE;
bHaltPulse := FALSE;

IF stCommand.rVelocity_rpm >= 0.0 THEN
    eVelocityDirection := MC_Positive_Direction;
ELSE
    eVelocityDirection := MC_Negative_Direction;
END_IF

IF bNewCommand THEN
    udiAcceptedCommandId := udiCommandId;
    bResetPulse := bDriveLinked AND stCommand.bReset;

    IF bDriveLinked AND stCommand.bStop THEN
        bHaltPulse := TRUE;
    ELSIF bDriveLinked AND stCommand.bEnable AND stCommand.bMoveVelocity THEN
        IF ABS(stCommand.rVelocity_rpm) > 0.0 THEN
            bSelectVelocityA := NOT bSelectVelocityA;
            bMoveVelocityPulseA := bSelectVelocityA;
            bMoveVelocityPulseB := NOT bSelectVelocityA;
        ELSE
            bHaltPulse := TRUE;
        END_IF
    END_IF
END_IF

(* 未完成真实驱动关联时Enable恒为FALSE，Torque只作为无效零值发布。 *)
fbPower(
    Axis := Axis,
    Enable := bDriveLinked AND stCommand.bEnable,
    Enable_Positive := bDriveLinked AND stCommand.bEnable,
    Enable_Negative := bDriveLinked AND stCommand.bEnable,
    Override := 100.0,
    BufferMode := MC_Aborting);
fbReset(Axis := Axis, Execute := bResetPulse);
fbMoveVelocityA(
    Axis := Axis,
    Execute := bMoveVelocityPulseA,
    Velocity := ABS(stCommand.rVelocity_rpm),
    Acceleration := ABS(stCommand.rAcceleration_rpm_s),
    Deceleration := ABS(stCommand.rDeceleration_rpm_s),
    Jerk := 0.0,
    Direction := eVelocityDirection,
    BufferMode := MC_Aborting);
fbMoveVelocityB(
    Axis := Axis,
    Execute := bMoveVelocityPulseB,
    Velocity := ABS(stCommand.rVelocity_rpm),
    Acceleration := ABS(stCommand.rAcceleration_rpm_s),
    Deceleration := ABS(stCommand.rDeceleration_rpm_s),
    Jerk := 0.0,
    Direction := eVelocityDirection,
    BufferMode := MC_Aborting);
fbHalt(
    Axis := Axis,
    Execute := bHaltPulse,
    Deceleration := ABS(stCommand.rDeceleration_rpm_s),
    Jerk := 0.0,
    BufferMode := MC_Aborting);

stStatus.bError := bDriveLinked AND (Axis.Status.Error OR fbPower.Error OR fbReset.Error
    OR fbMoveVelocityA.Error OR fbMoveVelocityB.Error OR fbHalt.Error);
stStatus.nErrorId := 0;
IF bDriveLinked AND Axis.Status.Error THEN
    stStatus.nErrorId := DWORD_TO_UDINT(Axis.NcToPlc.ErrorCode);
ELSIF fbPower.Error THEN
    stStatus.nErrorId := fbPower.ErrorID;
ELSIF fbReset.Error THEN
    stStatus.nErrorId := fbReset.ErrorID;
ELSIF fbMoveVelocityA.Error THEN
    stStatus.nErrorId := fbMoveVelocityA.ErrorID;
ELSIF fbMoveVelocityB.Error THEN
    stStatus.nErrorId := fbMoveVelocityB.ErrorID;
ELSIF fbHalt.Error THEN
    stStatus.nErrorId := fbHalt.ErrorID;
END_IF

stStatus.bReady := bDriveLinked AND fbPower.Status AND Axis.Status.Operational
    AND NOT stStatus.bError;
stStatus.bEnabled := bDriveLinked AND fbPower.Status;
stStatus.bMoving := bDriveLinked AND (Axis.Status.DiscreteMotion
    OR Axis.Status.ContinuousMotion);
stStatus.bStandstill := bDriveLinked AND Axis.Status.StandStill;
stStatus.bBusy := bDriveLinked AND (fbReset.Busy OR fbMoveVelocityA.Busy
    OR fbMoveVelocityB.Busy OR fbHalt.Busy);
stStatus.bDone := bDriveLinked AND (fbReset.Done OR fbMoveVelocityA.InVelocity
    OR fbMoveVelocityB.InVelocity OR fbHalt.Done);
stStatus.udiAcceptedCommandId := udiAcceptedCommandId;

IF bDriveLinked THEN
    stStatus.rActualVelocity_rpm := Axis.NcToPlc.ActVelo;
    stStatus.rActualTorque_Nm := Axis.NcToPlc.ActTorque;
ELSE
    stStatus.rActualVelocity_rpm := 0.0;
    stStatus.rActualTorque_Nm := 0.0;
END_IF;

END_FUNCTION_BLOCK

// ---- POUs/Fast/PRG_FastMonitoring.TcPOU
PROGRAM PRG_FastMonitoring
VAR
END_VAR

(* ---------------------------------------------------------
   程序骨架：快速过程统计、功率能量、窗口和曲线采样。
   所属任务：Task_CffFast，调用顺序4。
   唯一Owner：PRG_FastMonitoring。
   当前阶段：不记录生产结果，不执行字符串或文件操作。
   后续实现：只发布类型化监控结果和报警请求。
   --------------------------------------------------------- *)

END_PROGRAM

// ---- POUs/Main/PRG_ModeControl.TcPOU
PROGRAM PRG_ModeControl
VAR
END_VAR

(* ---------------------------------------------------------
   程序骨架：硬件模式与控制源权威输入仲裁。
   所属任务：Task_CffMain，调用顺序1。
   唯一Owner：PRG_ModeControl。
   当前阶段：不写入实际模式，不提供WPF旁路。
   后续实现：只允许冻结的三种Mode/Source组合。
   --------------------------------------------------------- *)

END_PROGRAM

// ---- POUs/Main/PRG_CommandDispatcher.TcPOU
PROGRAM PRG_CommandDispatcher
VAR
END_VAR

(* ---------------------------------------------------------
   程序骨架：HMI与Robot命令优先级、权限和事务仲裁。
   所属任务：Task_CffMain，调用顺序3。
   唯一Owner：PRG_CommandDispatcher。
   当前阶段：不产生Start/Stop/Initialize/Reset脉冲。
   后续实现：CommandId、Ack和单扫描内部Pulse。
   --------------------------------------------------------- *)

END_PROGRAM

// ---- POUs/Main/PRG_ProgramManager.TcPOU
PROGRAM PRG_ProgramManager
VAR
END_VAR

(* ---------------------------------------------------------
   程序骨架：焊接Program、版本、激活快照与Joining Point管理。
   所属任务：Task_CffMain，调用顺序4。
   唯一Owner：PRG_ProgramManager。
   当前阶段：不创建工艺参数，不激活任何Program。
   后续实现：Draft校验、Active快照和Revision。
   --------------------------------------------------------- *)

END_PROGRAM

// ---- POUs/Main/PRG_InitializeControl.TcPOU
PROGRAM PRG_InitializeControl
VAR
END_VAR

(* ---------------------------------------------------------
   程序骨架：设备初始化子状态机。
   所属任务：Task_CffMain，调用顺序5。
   唯一Owner：PRG_InitializeControl。
   当前阶段：不运动、不复位实际驱动、不伪造初始化完成。
   后续实现：Entry、Action、Success、Timeout和Fault。
   --------------------------------------------------------- *)

END_PROGRAM

// ---- POUs/Main/PRG_MaintenanceControl.TcPOU
PROGRAM PRG_MaintenanceControl
VAR
END_VAR

(* ---------------------------------------------------------
   程序骨架：Maintenance功能选择、Hold-to-Run和诊断权限。
   所属任务：Task_CffMain，调用顺序7。
   唯一Owner：PRG_MaintenanceControl。
   当前阶段：不输出点动、不绕过硬件绑定状态。
   后续实现：Heartbeat、SessionId和功能状态机。
   --------------------------------------------------------- *)

END_PROGRAM

// ---- POUs/Main/PRG_AutoControl.TcPOU
PROGRAM PRG_AutoControl
VAR
END_VAR

(* ---------------------------------------------------------
   程序骨架：Automatic+Robot生产循环编排。
   所属任务：Task_CffMain，调用顺序9。
   唯一Owner：PRG_AutoControl。
   当前阶段：生产硬件未绑定，Start权限保持关闭。
   后续实现：循环请求、完成握手和异常退出。
   --------------------------------------------------------- *)

END_PROGRAM

// ---- POUs/Main/PRG_FastenerControl.TcPOU
PROGRAM PRG_FastenerControl
VAR
END_VAR

(* ---------------------------------------------------------
   程序骨架：侦钉状态、请求和结果管理。
   所属任务：Task_CffMain，调用顺序10。
   唯一Owner：PRG_FastenerControl。
   当前阶段：不绑定传感器，不伪造Fastener OK。
   后续实现：状态机、超时、NOK和报警请求。
   --------------------------------------------------------- *)

END_PROGRAM

// ---- POUs/Main/PRG_FeederControl.TcPOU
PROGRAM PRG_FeederControl
VAR
END_VAR

(* ---------------------------------------------------------
   程序骨架：送料设备命令、状态和超时管理。
   所属任务：Task_CffMain，调用顺序11。
   唯一Owner：PRG_FeederControl。
   当前阶段：不绑定送料IO，不输出动作命令。
   后续实现：请求、完成、故障和恢复流程。
   --------------------------------------------------------- *)

END_PROGRAM

// ---- POUs/Main/PRG_AlarmControl.TcPOU
PROGRAM PRG_AlarmControl
VAR
END_VAR

(* ---------------------------------------------------------
   程序骨架：报警请求聚合、锁存、确认和复位。
   所属任务：Task_CffMain，调用顺序14。
   唯一Owner：PRG_AlarmControl。
   当前阶段：不生成安全合格声明，不替代人员安全系统。
   后续实现：AlarmCode、AlarmTextId、等级和时间戳。
   --------------------------------------------------------- *)

END_PROGRAM

// ---- POUs/Slow/PRG_Statistics.TcPOU
PROGRAM PRG_Statistics
VAR
END_VAR

(* ---------------------------------------------------------
   程序骨架：循环计数、NOK分类和过程统计发布。
   所属任务：Task_CffSlow，调用顺序3。
   唯一Owner：PRG_Statistics。
   当前阶段：无生产结果输入，不累加任何计数。
   后续实现：单一写入、复位权限和溢出处理。
   --------------------------------------------------------- *)

END_PROGRAM

// ---- POUs/Functions/FC_CalcEnergyIncrement.TcPOU
FUNCTION FC_CalcEnergyIncrement : LREAL
VAR_INPUT
    (* 本周期工程扭矩，单位牛米。 *)
    rTorque_Nm : LREAL;
    (* 本周期旋转速度，单位转每分钟。 *)
    rRpm : LREAL;
    (* 实际采样周期，单位秒。 *)
    rCycleTime_s : LREAL;
    (* TRUE时按功率绝对值累计能量。 *)
    bAbsolutePower : BOOL;
END_VAR
VAR_OUTPUT
    (* 周期为正且输入为有限工程值时为TRUE。 *)
    bValid : BOOL;
END_VAR
VAR
    (* 当前机械功率，单位瓦。 *)
    rPower_W : LREAL;
END_VAR

bValid := (rCycleTime_s > 0.0)
    AND FC_IsFiniteLReal(rValue := rTorque_Nm)
    AND FC_IsFiniteLReal(rValue := rRpm);
IF NOT bValid THEN
    FC_CalcEnergyIncrement := 0.0;
    RETURN;
END_IF

rPower_W := rTorque_Nm * FC_RpmToRadPerSec(rRpm := rRpm);
IF bAbsolutePower THEN
    rPower_W := ABS(rPower_W);
END_IF

(* 瓦乘秒得到本周期焦耳增量。 *)
FC_CalcEnergyIncrement := rPower_W * rCycleTime_s;

END_FUNCTION

// ---- POUs/Functions/FC_ConvertDirection.TcPOU
FUNCTION FC_ConvertDirection : LREAL
VAR_INPUT
    (* 需要按机械方向换算的工程值。 *)
    rValue : LREAL;
    (* 方向系数，只允许正一或负一。 *)
    nDirection : DINT;
END_VAR
VAR_OUTPUT
    (* 方向系数合法时为TRUE。 *)
    bValid : BOOL;
END_VAR

bValid := (nDirection = 1) OR (nDirection = -1);
IF bValid THEN
    FC_ConvertDirection := rValue * DINT_TO_LREAL(nDirection);
ELSE
    (* 非法方向不得静默放行，返回零并由调用者检查有效位。 *)
    FC_ConvertDirection := 0.0;
END_IF

END_FUNCTION

// ---- POUs/Functions/FC_Interpolate1D.TcPOU
FUNCTION FC_Interpolate1D : LREAL
VAR_INPUT
    (* 查询横坐标。 *)
    rX : LREAL;
    (* 第一个标定点横坐标。 *)
    rX0 : LREAL;
    (* 第一个标定点纵坐标。 *)
    rY0 : LREAL;
    (* 第二个标定点横坐标。 *)
    rX1 : LREAL;
    (* 第二个标定点纵坐标。 *)
    rY1 : LREAL;
    (* TRUE时禁止区间外外推。 *)
    bClampInput : BOOL;
END_VAR
VAR_OUTPUT
    (* 两个横坐标不重合且所有输入有限时为TRUE。 *)
    bValid : BOOL;
END_VAR
VAR
    (* 实际参与插值的横坐标。 *)
    rQueryX : LREAL;
END_VAR

bValid := (rX1 <> rX0)
    AND FC_IsFiniteLReal(rValue := rX)
    AND FC_IsFiniteLReal(rValue := rX0)
    AND FC_IsFiniteLReal(rValue := rY0)
    AND FC_IsFiniteLReal(rValue := rX1)
    AND FC_IsFiniteLReal(rValue := rY1);
IF NOT bValid THEN
    FC_Interpolate1D := rY0;
    RETURN;
END_IF

IF bClampInput THEN
    rQueryX := FC_ClampLReal(rValue := rX, rMinimum := rX0, rMaximum := rX1);
ELSE
    rQueryX := rX;
END_IF

FC_Interpolate1D := rY0 + ((rQueryX - rX0) / (rX1 - rX0)) * (rY1 - rY0);

END_FUNCTION

// ---- POUs/Functions/FC_CheckModeSourceMatrix.TcPOU
FUNCTION FC_CheckModeSourceMatrix : BOOL
VAR_INPUT
    (* 由硬件权威输入解析出的操作模式。 *)
    eOperationMode : E_OperationMode;
    (* 由硬件权威输入解析出的控制源。 *)
    eControlSource : E_ControlSource;
END_VAR

(* 只允许任务书冻结的三种模式与控制源组合。 *)
FC_CheckModeSourceMatrix :=
    ((eOperationMode = OP_MODE_MAINTENANCE) AND (eControlSource = CONTROL_SOURCE_LOCAL))
    OR ((eOperationMode = OP_MODE_MANUAL) AND (eControlSource = CONTROL_SOURCE_LOCAL))
    OR ((eOperationMode = OP_MODE_AUTOMATIC) AND (eControlSource = CONTROL_SOURCE_ROBOT));

END_FUNCTION

// ---- POUs/FunctionBlocks/Utility/FB_CommandHandshake.TcPOU
FUNCTION_BLOCK FB_CommandHandshake
VAR_INPUT
    (* 命令握手运行许可。 *)
    bEnable : BOOL;
    (* 握手状态复位请求；复位后接受编号回到零。 *)
    bReset : BOOL;
    (* 请求方最后完整写入的单调请求编号。 *)
    udiRequestId : UDINT;
END_VAR
VAR_OUTPUT
    (* 本实例已经原子接受的最后请求编号。 *)
    udiAcceptedId : UDINT;
    (* 本扫描发现并接受新请求时的单扫描脉冲。 *)
    bNewRequest : BOOL;
    (* 请求编号与已接受编号相同，表示重复请求。 *)
    bDuplicate : BOOL;
    (* 握手实例正在运行。 *)
    bValid : BOOL;
END_VAR

bNewRequest := FALSE;
bDuplicate := FALSE;
bValid := bEnable;

IF bReset THEN
    udiAcceptedId := 0;
    bValid := FALSE;
    RETURN;
END_IF

IF NOT bEnable OR (udiRequestId = 0) THEN
    RETURN;
END_IF

IF udiRequestId <> udiAcceptedId THEN
    (* 调用者必须在递增RequestId前写完其余邮箱字段。 *)
    udiAcceptedId := udiRequestId;
    bNewRequest := TRUE;
ELSE
    bDuplicate := TRUE;
END_IF

END_FUNCTION_BLOCK

// ---- POUs/FunctionBlocks/Utility/FB_AlarmLatch.TcPOU
FUNCTION_BLOCK FB_AlarmLatch
VAR_INPUT
    (* 报警锁存功能运行许可。 *)
    bEnable : BOOL;
    (* 操作者或上层状态机提出的复位请求。 *)
    bReset : BOOL;
    (* 本周期报警置位请求。 *)
    bSetRequest : BOOL;
    (* 产生报警的源条件当前仍然存在。 *)
    bSourceActive : BOOL;
    (* 当前模式、权限和状态允许清除锁存。 *)
    bResetAllowed : BOOL;
END_VAR
VAR_OUTPUT
    (* 报警已经锁存；源条件消失后仍保持。 *)
    bLatched : BOOL;
    (* 报警首次置位的单扫描脉冲。 *)
    bSetPulse : BOOL;
    (* 复位请求因源仍存在或权限不足被拒绝。 *)
    bResetRejected : BOOL;
    (* 报警锁存功能处于运行状态。 *)
    bValid : BOOL;
END_VAR
VAR
    (* 上一扫描的置位请求，用于形成边沿脉冲。 *)
    bPreviousSetRequest : BOOL;
END_VAR

bSetPulse := FALSE;
bResetRejected := FALSE;
bValid := bEnable;

IF NOT bEnable THEN
    bPreviousSetRequest := bSetRequest;
    RETURN;
END_IF

(* 置位优先于复位，确保同一扫描出现故障时不会被清除。 *)
IF bSetRequest OR bSourceActive THEN
    bSetPulse := NOT bLatched AND ((bSetRequest AND NOT bPreviousSetRequest) OR bSourceActive);
    bLatched := TRUE;
    IF bReset THEN
        (* 故障源仍存在或同一扫描重新置位时，复位请求明确被拒绝。 *)
        bResetRejected := TRUE;
    END_IF
ELSIF bReset THEN
    IF bResetAllowed AND NOT bSourceActive THEN
        bLatched := FALSE;
    ELSE
        bResetRejected := TRUE;
    END_IF
END_IF

bPreviousSetRequest := bSetRequest;

END_FUNCTION_BLOCK
